ABB RobotStudio station: jaffir welding robot.rsstn

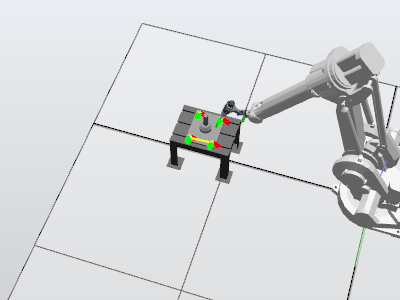
Station Station (saved by RobotStudio 22.3.10141.1)
Controller Controller42
  mechanical unit ROB_1: IRB1410_5_144__01, 6 joints, base frame (0, 0, 0) mm
Layout (positions relative to the parent item):
  - IRB1410_5_144__01 [mechanism, from Robots\IRB1410_5_144_G_01.rslib] at (0, 0, 0) mm; joint values [-0.0971, 0.3098, 0.9519, -0.1229, -0.3917, 0.1365] (rad or m)
  - MyTool [mechanism, from Training Objects\myTool.rslib] at (916.21, -85.25, 484.28) mm, rotated rx 175.26 ry 57.66 rz 172 deg
  - table_and_fixture_140 [part, from Training Objects\propeller_table.rslib] at (938.29, -175, 0) mm
Attachment: MyTool is attached to IRB1410_5_144__01 / Link6
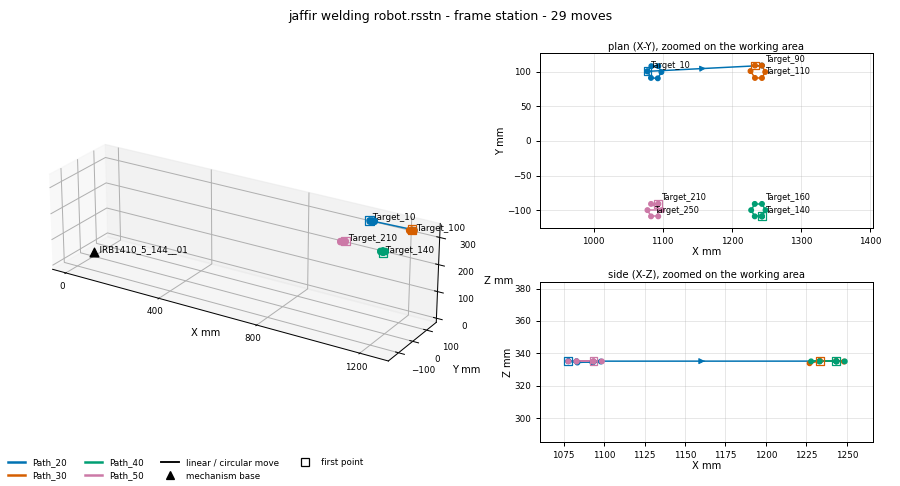
[picture p0: tool path of jaffir welding robot.rsstn in frame station, 29 of 29 moves have a stored position in this frame; points joined in program order, loops and branches not executed]
Targets, tools, work objects and paths stored in the station, written as RAPID:
! task T_ROB1
MODULE CalibData
  PERS tooldata MyTool:=[TRUE,[[31.792631019,0,229.638935148],[0.945518576,0,0.325568154,0]],[1,[0,0,1],[1,0,0,0],0,0,0]];
ENDMODULE

! task T_ROB1
MODULE Module1
  CONST robtarget Target_10:=[[1077.962038824,100.705302487,335.12969921],[0.172134531,0.03808925,0.984209903,0.015804386],[0,0,-1,0],[9E+09,9E+09,9E+09,9E+09,9E+09,9E+09]];
  CONST robtarget Target_20:=[[1083.530992517,108.208893772,334.277868454],[0.172133731,0.038089246,0.984210043,0.015804393],[0,0,-1,0],[9E+09,9E+09,9E+09,9E+09,9E+09,9E+09]];
  CONST robtarget Target_30:=[[1093.62399946,108.208893751,334.792272818],[0.172133633,0.038089261,0.98421006,0.015804404],[0,0,-1,0],[9E+09,9E+09,9E+09,9E+09,9E+09,9E+09]];
  CONST robtarget Target_40:=[[1098.062977175,99.720254401,334.900175477],[0.17213274,0.038089257,0.984210216,0.015804423],[0,0,-1,0],[9E+09,9E+09,9E+09,9E+09,9E+09,9E+09]];
  CONST robtarget Target_60:=[[1092.844024925,90.61931941,334.275196894],[0.172130842,0.038089215,0.984210549,0.015804416],[0,0,-1,0],[9E+09,9E+09,9E+09,9E+09,9E+09,9E+09]];
  CONST robtarget Target_70:=[[1083.011990832,91.235942678,335.113279055],[0.172130355,0.038089205,0.984210634,0.015804446],[0,0,-1,0],[9E+09,9E+09,9E+09,9E+09,9E+09,9E+09]];
  CONST robtarget Target_80:=[[1233.378043693,109.127307201,335.150393613],[0.172129048,0.0380892,0.984210862,0.015804489],[0,0,-1,0],[9E+09,9E+09,9E+09,9E+09,9E+09,9E+09]];
  CONST robtarget Target_90:=[[1243.407007815,109.127297101,335.150374945],[0.172128958,0.038089197,0.984210878,0.015804491],[0,0,-1,0],[9E+09,9E+09,9E+09,9E+09,9E+09,9E+09]];
  CONST robtarget Target_100:=[[1248.190976865,99.842238986,334.848681331],[0.172128645,0.03808919,0.984210933,0.015804503],[0,0,-1,0],[9E+09,9E+09,9E+09,9E+09,9E+09,9E+09]];
  CONST robtarget Target_110:=[[1243.487943545,91.089442246,335.299188344],[0.172127556,0.03808915,0.984211125,0.015804512],[0,0,-1,0],[9E+09,9E+09,9E+09,9E+09,9E+09,9E+09]];
  CONST robtarget Target_120:=[[1233.383057426,91.178670916,335.299192982],[0.172127459,0.038089135,0.984211143,0.015804511],[0,0,-1,0],[9E+09,9E+09,9E+09,9E+09,9E+09,9E+09]];
  CONST robtarget Target_130:=[[1226.964939159,101.090788976,333.832789731],[0.172127352,0.038089148,0.98421116,0.015804549],[0,0,-1,0],[9E+09,9E+09,9E+09,9E+09,9E+09,9E+09]];
  CONST robtarget Target_140:=[[1243.489013888,-108.999995295,334.999995516],[0.172122841,0.038089098,0.98421195,0.015804602],[-1,-1,0,0],[9E+09,9E+09,9E+09,9E+09,9E+09,9E+09]];
  CONST robtarget Target_150:=[[1248.684986209,-100.00000144,335.000000853],[0.172122746,0.038089098,0.984211967,0.015804602],[-1,-1,0,0],[9E+09,9E+09,9E+09,9E+09,9E+09,9E+09]];
  CONST robtarget Target_160:=[[1243.489012556,-91.000000276,334.999995579],[0.17212254,0.0380891,0.984212003,0.015804601],[-1,-1,0,0],[9E+09,9E+09,9E+09,9E+09,9E+09,9E+09]];
  CONST robtarget Target_170:=[[1233.09602373,-90.999995094,335.000018452],[0.172122456,0.038089101,0.984212017,0.015804603],[-1,-1,0,0],[9E+09,9E+09,9E+09,9E+09,9E+09,9E+09]];
  CONST robtarget Target_180:=[[1227.900032116,-99.999997492,335.000015262],[0.172122367,0.038089101,0.984212033,0.015804604],[-1,-1,0,0],[9E+09,9E+09,9E+09,9E+09,9E+09,9E+09]];
  CONST robtarget Target_190:=[[1233.095985357,-108.999996407,334.999983915],[0.172122349,0.038089101,0.984212036,0.015804602],[-1,-1,0,0],[9E+09,9E+09,9E+09,9E+09,9E+09,9E+09]];
  CONST robtarget Target_200:=[[1243.489036222,-108.999999573,335.000000831],[0.172122259,0.038089098,0.984212052,0.0158046],[-1,-1,0,0],[9E+09,9E+09,9E+09,9E+09,9E+09,9E+09]];
  CONST robtarget Target_210:=[[1093.489048762,-90.999999306,335.000002237],[0.172122152,0.038089103,0.98421207,0.015804612],[-1,-1,0,0],[9E+09,9E+09,9E+09,9E+09,9E+09,9E+09]];
  CONST robtarget Target_220:=[[1083.096038367,-90.999996034,335.000000228],[0.172122157,0.0380891,0.98421207,0.015804612],[-1,-1,0,0],[9E+09,9E+09,9E+09,9E+09,9E+09,9E+09]];
  CONST robtarget Target_230:=[[1098.685030257,-99.999996549,335.000008817],[0.172122154,0.038089099,0.98421207,0.015804612],[-1,-1,0,0],[9E+09,9E+09,9E+09,9E+09,9E+09,9E+09]];
  CONST robtarget Target_240:=[[1077.900059604,-99.999997379,334.999999313],[0.172122153,0.038089101,0.98421207,0.015804612],[-1,-1,0,0],[9E+09,9E+09,9E+09,9E+09,9E+09,9E+09]];
  CONST robtarget Target_250:=[[1083.096032332,-108.999999259,334.999994155],[0.172122149,0.038089103,0.984212071,0.015804613],[-1,-1,0,0],[9E+09,9E+09,9E+09,9E+09,9E+09,9E+09]];
  CONST robtarget Target_260:=[[1093.489051174,-108.999998612,335.000005599],[0.172122135,0.038089104,0.984212073,0.015804614],[-1,-1,0,0],[9E+09,9E+09,9E+09,9E+09,9E+09,9E+09]];
  PROC Path_20()
    MoveL Target_10,v1000,fine,MyTool\WObj:=wobj0;
    MoveL Target_20,v1000,fine,MyTool\WObj:=wobj0;
    MoveL Target_30,v1000,fine,MyTool\WObj:=wobj0;
    MoveL Target_40,v1000,fine,MyTool\WObj:=wobj0;
    MoveL Target_60,v1000,fine,MyTool\WObj:=wobj0;
    MoveL Target_70,v1000,fine,MyTool\WObj:=wobj0;
    MoveL Target_10,v1000,fine,MyTool\WObj:=wobj0;
    MoveL Target_90,v1000,fine,MyTool\WObj:=wobj0;
  ENDPROC
  PROC Path_30()
    MoveL Target_80,v1000,fine,MyTool\WObj:=wobj0;
    MoveL Target_90,v1000,fine,MyTool\WObj:=wobj0;
    MoveL Target_100,v1000,fine,MyTool\WObj:=wobj0;
    MoveL Target_110,v1000,fine,MyTool\WObj:=wobj0;
    MoveL Target_120,v1000,fine,MyTool\WObj:=wobj0;
    MoveL Target_130,v1000,fine,MyTool\WObj:=wobj0;
  ENDPROC
  PROC Path_40()
    MoveL Target_140,v1000,fine,MyTool\WObj:=wobj0;
    MoveL Target_150,v1000,fine,MyTool\WObj:=wobj0;
    MoveL Target_160,v1000,fine,MyTool\WObj:=wobj0;
    MoveL Target_170,v1000,fine,MyTool\WObj:=wobj0;
    MoveL Target_180,v1000,fine,MyTool\WObj:=wobj0;
    MoveL Target_190,v1000,fine,MyTool\WObj:=wobj0;
    MoveL Target_200,v1000,fine,MyTool\WObj:=wobj0;
    MoveL Target_140,v1000,fine,MyTool\WObj:=wobj0;
  ENDPROC
  PROC Path_50()
    MoveL Target_210,v1000,fine,MyTool\WObj:=wobj0;
    MoveL Target_220,v1000,fine,MyTool\WObj:=wobj0;
    MoveL Target_230,v1000,fine,MyTool\WObj:=wobj0;
    MoveL Target_240,v1000,fine,MyTool\WObj:=wobj0;
    MoveL Target_250,v1000,fine,MyTool\WObj:=wobj0;
    MoveL Target_260,v1000,fine,MyTool\WObj:=wobj0;
    MoveL Target_210,v1000,fine,MyTool\WObj:=wobj0;
  ENDPROC
ENDMODULE

